Omron Sysmac Studio project ScaleTrans (Sysmac Studio 1.65.0.64007, StandardProject)

# Controller new_Controller_0: NX1P2-1040DT1 version 1.69
Task PrimaryTask (priority 4, period or condition 2000): Program0



PROGRAM Program0
VAR
    A_IN : REAL;
    A_X0 : REAL;
    A_Y0 : REAL;
    A_X1 : REAL;
    A_Y1 : REAL;
    A_OUT : REAL;
    temppp : REAL;
END_VAR

(* Section Section0: ladder, written here as Structured Text *)

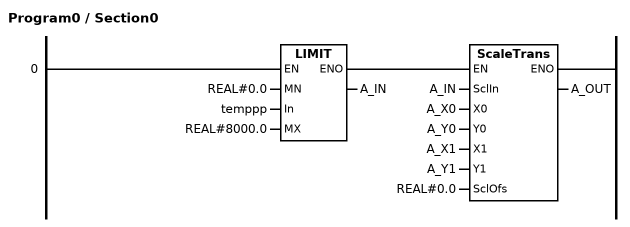
(* Rung 0 *)
A_IN := LIMIT(MN := REAL#0.0, In := temppp, MX := REAL#8000.0);
A_OUT := ScaleTrans(SclIn := A_IN, X0 := A_X0, Y0 := A_Y0, X1 := A_X1, Y1 := A_Y1, SclOfs := REAL#0.0);
END_PROGRAM